// SIMATIC S7-200 project (STEP 7-Micro/WIN), CPU 224XP REL 02.01

SYMBOL_TABLE USUARIO1
CAFE_SOLO        I0.0
CAFE_EXPRESO     I0.1
C_LECHE          I0.2
LECHE            I0.3
TE               I0.4
AGUA             I0.5
P_MONEDERO       I0.6
EV_CAFE          Q0.0
EV_LECHE         Q0.1
EV_AGUA          Q0.2
EV_TE            Q0.3
CONTADOR         MW4
SEGURIDAD        Q2.0
SELECCION        Q2.1
AUX_SOLO         Q2.2
AUX_EXPRESSO     Q2.3
AUX_CCL          Q2.4
AUX_LECHE        Q2.5
AUX_TE           Q2.6
AUX_AGUA         Q2.7
END_SYMBOL_TABLE

ORGANIZATION_BLOCK PRINCIPAL:OB1
TITLE=COMENTARIOS DEL PROGRAMA
BEGIN
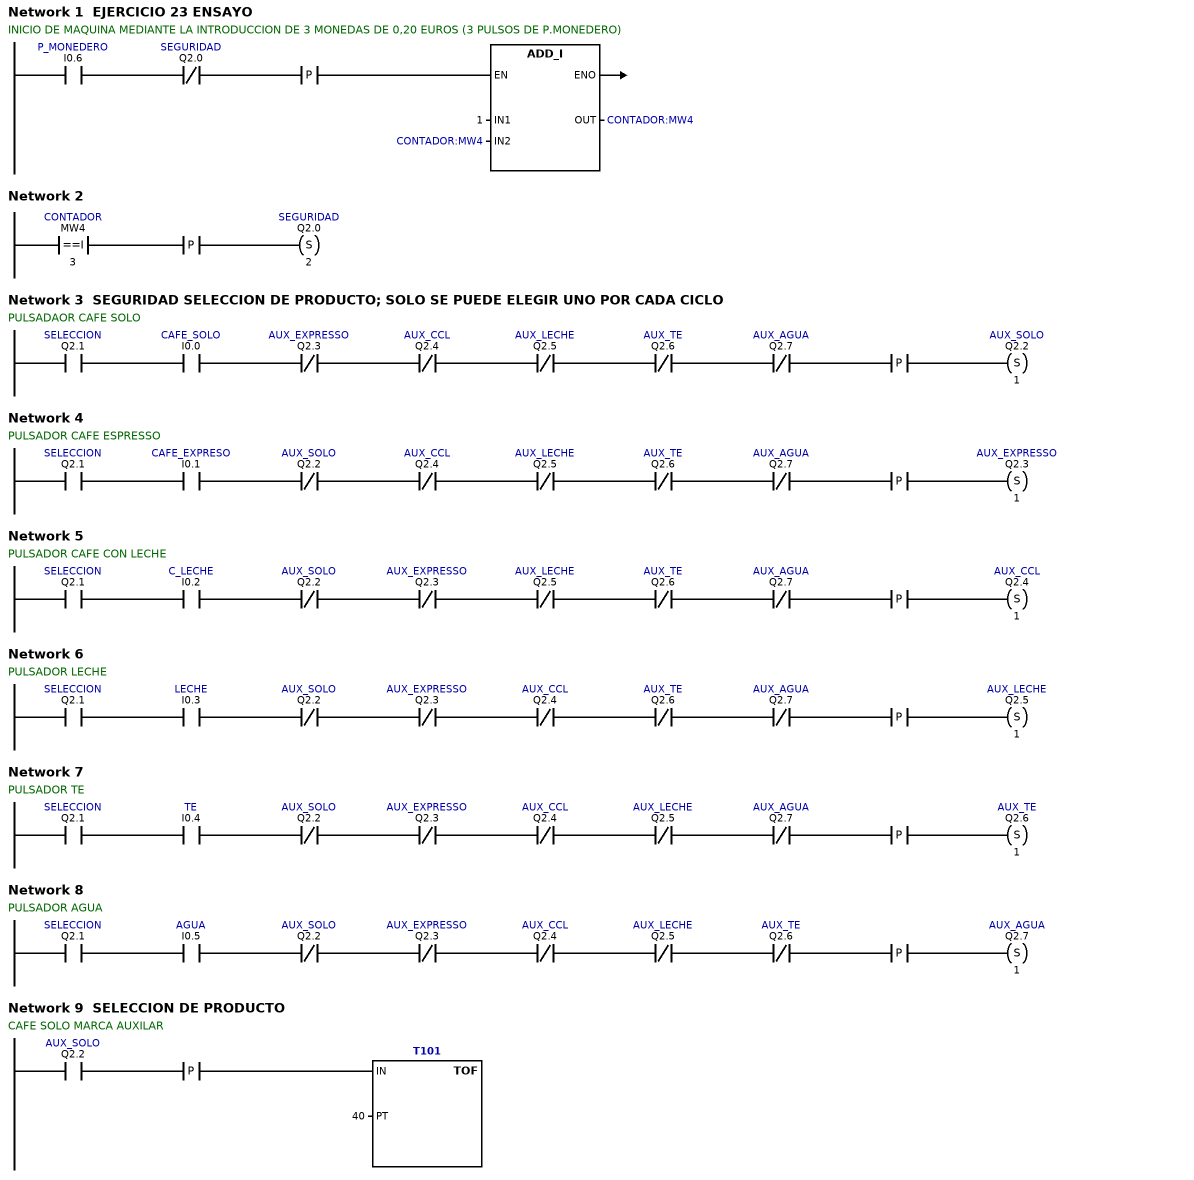
Network 1 // EJERCICIO 23 ENSAYO
// INICIO DE MAQUINA MEDIANTE LA INTRODUCCION DE 3 MONEDAS DE 0,20 EUROS (3 PULSOS DE P.MONEDERO)
LD     P_MONEDERO:I0.6
AN     SEGURIDAD:Q2.0
EU
+I     1, CONTADOR:MW4
Network 2
LDW=   CONTADOR:MW4, 3
EU
S      SEGURIDAD:Q2.0, 2
Network 3 // SEGURIDAD SELECCION DE PRODUCTO; SOLO SE PUEDE ELEGIR UNO POR CADA CICLO
// PULSADAOR CAFE SOLO
LD     SELECCION:Q2.1
A      CAFE_SOLO:I0.0
AN     AUX_EXPRESSO:Q2.3
AN     AUX_CCL:Q2.4
AN     AUX_LECHE:Q2.5
AN     AUX_TE:Q2.6
AN     AUX_AGUA:Q2.7
EU
S      AUX_SOLO:Q2.2, 1
Network 4
// PULSADOR CAFE ESPRESSO
LD     SELECCION:Q2.1
A      CAFE_EXPRESO:I0.1
AN     AUX_SOLO:Q2.2
AN     AUX_CCL:Q2.4
AN     AUX_LECHE:Q2.5
AN     AUX_TE:Q2.6
AN     AUX_AGUA:Q2.7
EU
S      AUX_EXPRESSO:Q2.3, 1
Network 5
// PULSADOR CAFE CON LECHE
LD     SELECCION:Q2.1
A      C_LECHE:I0.2
AN     AUX_SOLO:Q2.2
AN     AUX_EXPRESSO:Q2.3
AN     AUX_LECHE:Q2.5
AN     AUX_TE:Q2.6
AN     AUX_AGUA:Q2.7
EU
S      AUX_CCL:Q2.4, 1
Network 6
// PULSADOR LECHE
LD     SELECCION:Q2.1
A      LECHE:I0.3
AN     AUX_SOLO:Q2.2
AN     AUX_EXPRESSO:Q2.3
AN     AUX_CCL:Q2.4
AN     AUX_TE:Q2.6
AN     AUX_AGUA:Q2.7
EU
S      AUX_LECHE:Q2.5, 1
Network 7
// PULSADOR TE
LD     SELECCION:Q2.1
A      TE:I0.4
AN     AUX_SOLO:Q2.2
AN     AUX_EXPRESSO:Q2.3
AN     AUX_CCL:Q2.4
AN     AUX_LECHE:Q2.5
AN     AUX_AGUA:Q2.7
EU
S      AUX_TE:Q2.6, 1
Network 8
// PULSADOR AGUA
LD     SELECCION:Q2.1
A      AGUA:I0.5
AN     AUX_SOLO:Q2.2
AN     AUX_EXPRESSO:Q2.3
AN     AUX_CCL:Q2.4
AN     AUX_LECHE:Q2.5
AN     AUX_TE:Q2.6
EU
S      AUX_AGUA:Q2.7, 1
Network 9 // SELECCION DE PRODUCTO
//   CAFE SOLO MARCA AUXILAR
LD     AUX_SOLO:Q2.2
EU
TOF    T101, 40
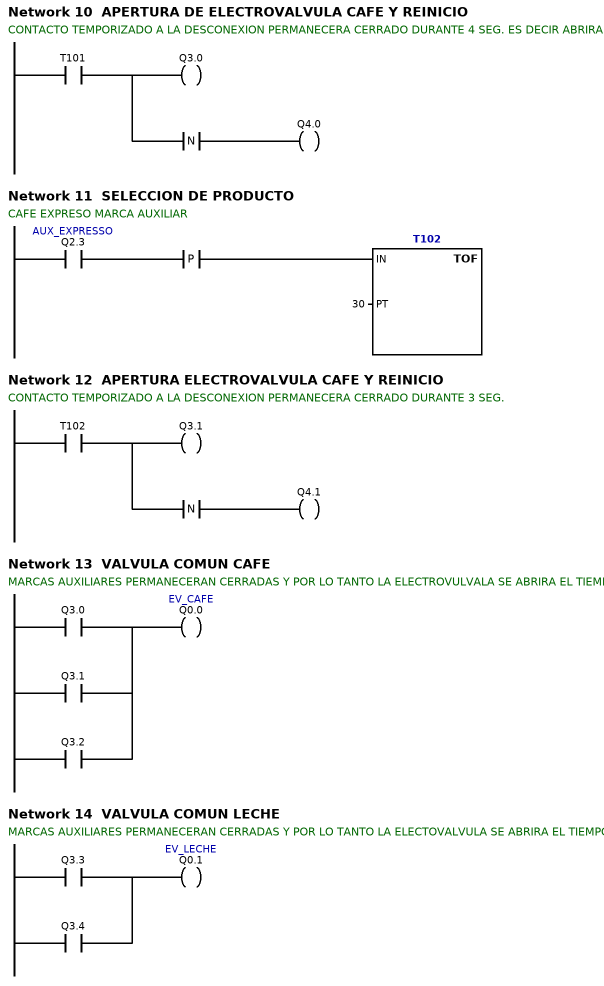
Network 10 // APERTURA DE ELECTROVALVULA CAFE Y REINICIO
// CONTACTO TEMPORIZADO A LA DESCONEXION PERMANECERA CERRADO DURANTE 4 SEG. ES DECIR ABRIRA LA ELECTOVALVULA DURANTE ESE TIEMPO
LD     T101
=      Q3.0
ED
=      Q4.0
Network 11 // SELECCION DE PRODUCTO
//  CAFE EXPRESO MARCA AUXILIAR
LD     AUX_EXPRESSO:Q2.3
EU
TOF    T102, 30
Network 12 // APERTURA ELECTROVALVULA CAFE Y REINICIO
// CONTACTO TEMPORIZADO A LA DESCONEXION PERMANECERA CERRADO DURANTE 3 SEG.
LD     T102
=      Q3.1
ED
=      Q4.1
Network 13 // VALVULA COMUN CAFE
// MARCAS AUXILIARES PERMANECERAN CERRADAS Y POR LO TANTO LA ELECTROVULVALA SE ABRIRA EL TIEMPO CORRESPONDIENTE A CADA PRODUCTO
LD     Q3.0
O      Q3.1
O      Q3.2
=      EV_CAFE:Q0.0
Network 14 // VALVULA COMUN LECHE
// MARCAS AUXILIARES PERMANECERAN CERRADAS Y POR LO TANTO LA ELECTOVALVULA SE ABRIRA EL TIEMPO CORRESPONDIENTE CADA PRODUCTO
LD     Q3.3
O      Q3.4
=      EV_LECHE:Q0.1
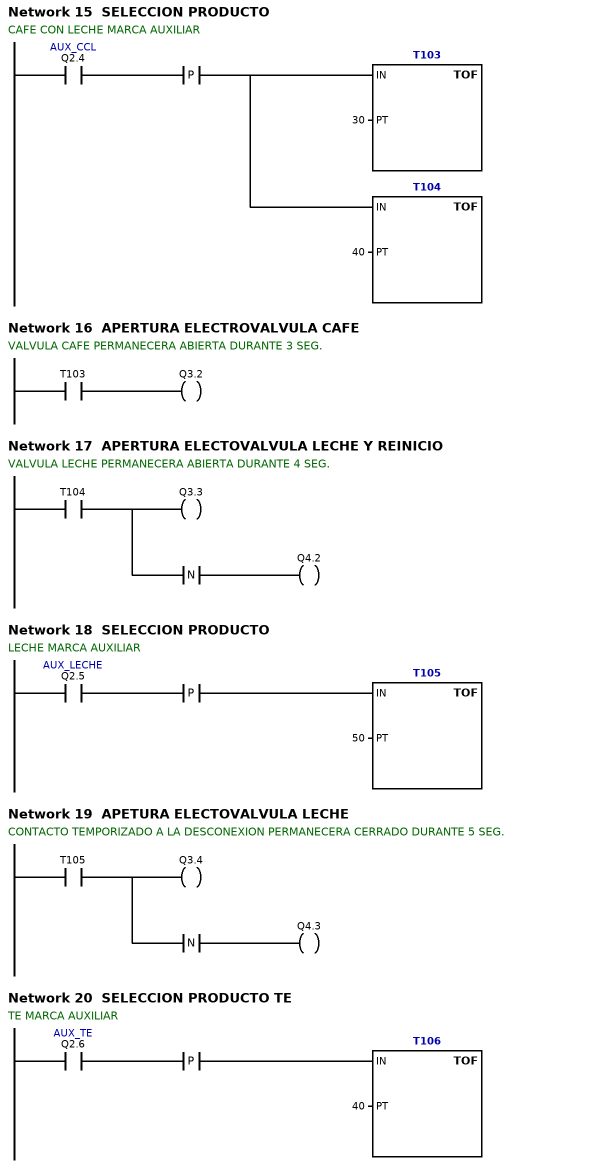
Network 15 // SELECCION PRODUCTO 
//  CAFE CON LECHE MARCA AUXILIAR 
LD     AUX_CCL:Q2.4
EU
TOF    T103, 30
TOF    T104, 40
Network 16 // APERTURA ELECTROVALVULA CAFE
// VALVULA CAFE PERMANECERA ABIERTA DURANTE 3 SEG.
LD     T103
=      Q3.2
Network 17 // APERTURA ELECTOVALVULA LECHE Y REINICIO
// VALVULA LECHE PERMANECERA ABIERTA DURANTE 4 SEG.
LD     T104
=      Q3.3
ED
=      Q4.2
Network 18 // SELECCION PRODUCTO
//   LECHE MARCA AUXILIAR 
LD     AUX_LECHE:Q2.5
EU
TOF    T105, 50
Network 19 // APETURA ELECTOVALVULA LECHE
// CONTACTO TEMPORIZADO A LA DESCONEXION PERMANECERA CERRADO DURANTE 5 SEG.
LD     T105
=      Q3.4
ED
=      Q4.3
Network 20 // SELECCION PRODUCTO TE
//  TE MARCA AUXILIAR 
LD     AUX_TE:Q2.6
EU
TOF    T106, 40
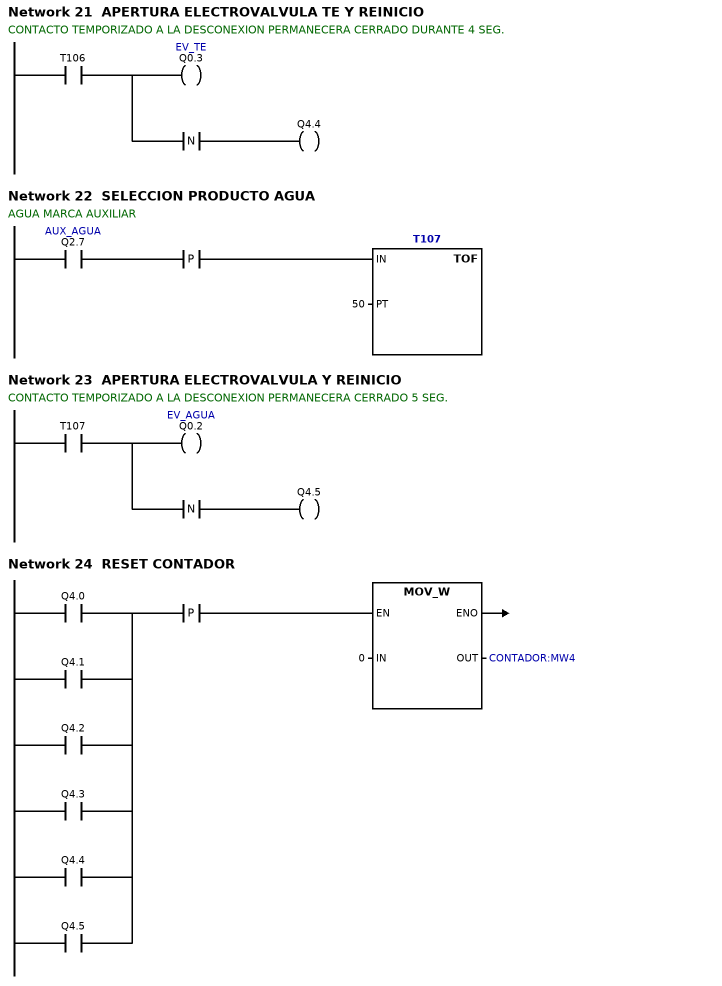
Network 21 // APERTURA ELECTROVALVULA TE Y REINICIO
// CONTACTO TEMPORIZADO A LA DESCONEXION PERMANECERA CERRADO DURANTE 4 SEG.
LD     T106
=      EV_TE:Q0.3
ED
=      Q4.4
Network 22 // SELECCION PRODUCTO AGUA
// AGUA MARCA AUXILIAR
LD     AUX_AGUA:Q2.7
EU
TOF    T107, 50
Network 23 // APERTURA ELECTROVALVULA Y REINICIO
// CONTACTO TEMPORIZADO A LA DESCONEXION PERMANECERA CERRADO 5 SEG.
LD     T107
=      EV_AGUA:Q0.2
ED
=      Q4.5
Network 24 // RESET CONTADOR
LD     Q4.0
O      Q4.1
O      Q4.2
O      Q4.3
O      Q4.4
O      Q4.5
EU
MOVW   0, CONTADOR:MW4
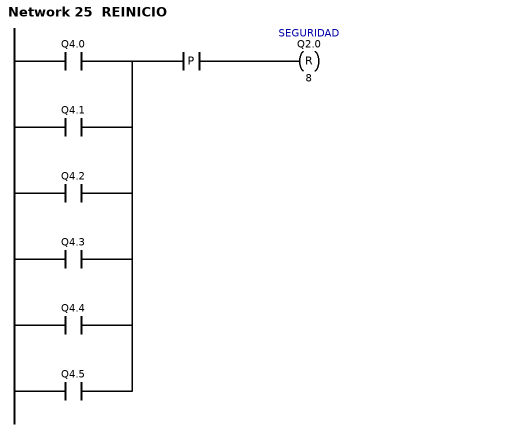
Network 25 // REINICIO
LD     Q4.0
O      Q4.1
O      Q4.2
O      Q4.3
O      Q4.4
O      Q4.5
EU
R      SEGURIDAD:Q2.0, 8
END_ORGANIZATION_BLOCK
